FUNCTION_BLOCK ABSTRACT RFC_MoveWorkpiece_Base EXTENDS ControlPrimitiveBase
VAR_INPUT
END_VAR
VAR_OUTPUT
END_VAR
VAR
	m_ptrRFC: POINTER TO RefeedingConveyor;
	
	m_step: INT := 0;
END_VAR

SUPER^();

METHOD  Abort : BOOL
VAR_INPUT
END_VAR
m_ptrRFC^.METH_ConveyorStop();
m_ptrRFC^.METH_Switch_Retract();
Abort := TRUE;
END_METHOD

METHOD PROTECTED ABSTRACT AtTarget : BOOL
VAR_INPUT
END_VAR
END_METHOD

(* Execution logic of this Control Primitive. *)
METHOD PROTECTED ExecuteInternal : BOOL
VAR_INPUT
	i_params: ParameterSet;
END_VAR
CASE m_step OF
	0: // to target	
	IF NOT AtTarget() THEN
		m_ptrRFC^.METH_ConveyorForward();
		m_step := 1;
	END_IF
		
	1:
	IF AtTarget() THEN
		m_ptrRFC^.METH_ConveyorStop();
		//m_ptrPAC^.METH_Switch_Extend();
		m_step := 0;
		ExecuteInternal := TRUE;
	END_IF
		
END_CASE
END_METHOD

END_FUNCTION_BLOCK

(* stored: Version 1.1.0.1, ProductVersion 3.1.4024.12
   POU RFC_MoveWorkpiece_Base: Id {5cee6e47-6f21-4489-a7df-606755c33154}, SpecialFunc None
   Method Abort: Id {f3d32937-611f-4c2e-a5a8-8806523bfd8d}
   Method AtTarget: Id {6aebcdf5-b8e3-42f6-bd5c-f7cf29a66099}
   Method ExecuteInternal: Id {bb7180ca-bcc1-4a35-a753-f4929dce7c7a} *)
